(* Logix 5000 project; controller GolfBall vendor 1 type 14 code 149 rev 36.12; software revision 36.03 *)

TASK MainTask (continuous, watchdog 500 ms) : MainProgram

MODULES
   Local : vendor 1 type 14 code 149 (Compact 0, rev 36.12)
       : 1769-IQ16 (Compact 2, rev 1.1, Input RPI 20 ms)
       : 1769-IQ16 (Compact 3, rev 3.1, Input RPI 20 ms)
      Relay : 1769-OB16 (Compact 4, rev 3.1, Output RPI 20 ms)
      Discrete_IO : Embedded (Compact 1, rev 3.1, Output RPI 20 ms)
END_MODULES

TYPE FAULTRECORD :   // Stores the MajorFaultRecord attribute or MinorFaultRecord attribute of the Program object
STRUCT
   Time_Low : DINT;   // Lower 32 bits of the fault timestamp value
   Time_High : DINT;   // Upper 32 bits of the fault timestamp value
   Type : INT;   // Fault type (program, I/O, and so forth)
   Code : INT;   // Unique code for the fault
   Info : DINT[8];   // Fault specific information
END_STRUCT
END_TYPE

VAR_GLOBAL   (* controller tags *)
   Actuate_T1_Diverter : ALIAS FOR Local:4:O.Data.5; {access Read Only}
   Actuate_T1_Drop_Advance : ALIAS FOR Local:4:O.Data.12; {access Read Only}
   Actuate_T1_Drop_Release : ALIAS FOR Local:4:O.Data.13; {access Read Only}
   Actuate_T2_Diverter : ALIAS FOR Local:4:O.Data.6; {access Read Only}
   Actuate_T2_Drop_Advance : ALIAS FOR Local:4:O.Data.10; {access Read Only}
   Actuate_T2_Drop_Release : ALIAS FOR Local:4:O.Data.11; {access Read Only}
   Actuate_T3_Diverter : ALIAS FOR Local:4:O.Data.7; {access Read Only}
   Actuate_T3_Drop_Advance : ALIAS FOR Local:4:O.Data.8; {access Read Only}
   Actuate_T3_Drop_Release : ALIAS FOR Local:4:O.Data.9; {access Read Only}
   All_Tubes_Full : BOOL; {access Read Only}
   Auto_Run_Enable : BOOL; {access Read Only}
   Ball_Bypass_Photo : ALIAS FOR Local:1:I.Data.3; {access Read Only}
   Ball_Feeder_Extended : ALIAS FOR Local:3:I.Data.8; {access Read Only}
   Ball_Feeder_Intermediate : ALIAS FOR Local:3:I.Data.9; {access Read Only}
   Ball_Feeder_Retracted : ALIAS FOR Local:3:I.Data.10; {access Read Only}
   Ball_Feeder_Retracted_Timer : FBD_TIMER := (PRE := 400, Reset := 1); {access Read Only}
   Ball_Feeder_Step : DINT; {access Read Only}
   Ball_Present_Ball_Feeder : ALIAS FOR Local:3:I.Data.11; {access Read Only}
   Blink_Bit : BOOL; {access Read Only}
   Color : DINT; {access Read Only}
   Color_Advance_Cylinder_Extended : ALIAS FOR Local:1:I.Data.6; {access Read Only}
   Color_Advance_Cylinder_Retracted : ALIAS FOR Local:1:I.Data.7; {access Read Only}
   Color_Read_Advance_Cylinder_Timer : FBD_TIMER := (PRE := 1000); {access Read Only}
   Color_Read_Dwell_Timer : FBD_TIMER := (PRE := 1500); {access Read Only}
   Color_Release_Cylinder_Extended : ALIAS FOR Local:1:I.Data.8; {access Read Only}
   Color_Release_Cylinder_Retracted : ALIAS FOR Local:1:I.Data.9; {access Read Only}
   Color_Scan_Green : ALIAS FOR Local:3:I.Data.13; {access Read Only}
   Color_Scan_Orange : ALIAS FOR Local:3:I.Data.14; {access Read Only}
   Color_Scan_Pink : ALIAS FOR Local:3:I.Data.12; {access Read Only}
   Color_Sort_Dwell_Timer : FBD_TIMER := (TimerEnable := 1, PRE := 3500, ACC := 651, EN := 1, TT := 1); {access Read Only}
   Color_Sort_Step : DINT; {access Read Only}
   Drop_Ball_Feeder : ALIAS FOR Local:4:O.Data.15; {access Read Only}
   Dropping_Ball_Feeder : BOOL; {access Read Only}
   Fault : BOOL; {access Read Only}   // Master Fault
   Fault_Blink : BOOL; {access Read Only}
   Fault_Feeder_Drop_Timeout : BOOL; {access Read Only}
   Fault_Feeder_Lift_Timeout : BOOL; {access Read Only}
   Fault_Feeder_Watchdog : BOOL; {access Read Only}
   Feed_Bypass : BOOL; {access Read Only}
   Feed_Resume_OS : BOOL; {access Read Only}
   Feed_Resume_Storage : BOOL; {access Read Only}
   Feed_Run : BOOL; {access Read Only}
   Feeder_Drop_Timeout_Timer : FBD_TIMER := (PRE := 3000, Reset := 1); {access Read Only}
   Feeder_Extend_Count : DINT; {access Read Only}
   Feeder_Fault : BOOL; {access Read Only}
   Feeder_Fault_Active : BOOL; {access Read Only}
   Feeder_Hard_Fault_HMI : BOOL; {access Read Only}
   Feeder_Homing : BOOL; {access Read Only}
   Feeder_Lift_Timeout_Timer : FBD_TIMER := (TimerEnable := 1, PRE := 3000, ACC := 3000, EN := 1, DN := 1); {access Read Only}
   Feeder_Motion_Detected_OS : BOOL; {access Read Only}
   Feeder_Motion_Storage : BOOL; {access Read Only}
   Feeder_Recovery_Attempt_Counter : DINT; {access Read Only}
   Feeder_Recovery_Timer : FBD_TIMER := (PRE := 5000); {access Read Only}
   Feeder_Recovery_Total : DINT; {access Read Only}
   Feeder_Stuck_at_Sensor : BOOL; {access Read Only}
   Feeder_Watchdog_Timer : FBD_TIMER := (TimerEnable := 1, PRE := 5000, ACC := 3002, EN := 1, TT := 1); {access Read Only}
   Fill_Indexes_Cleared : BOOL := 1; {access Read Only}
   Green : DINT := 3; {access Read Only}
   HMI_All_Tubes_Are_Empty : INT := 10;
   HMI_ColorStationAdv : BOOL;
   HMI_ColorStationRel : BOOL := 1;
   HMI_Diverter1 : BOOL;
   HMI_Diverter2 : BOOL;
   HMI_Diverter3 : BOOL;
   HMI_DropFeedCylinder : BOOL;
   HMI_Fault_Reset_PB : BOOL;
   HMI_Page_State : INT := 2;
   HMI_RaiseFeedCylinder : BOOL;
   HMI_RequestedMode : INT;   // 30: Auto 20: Manual 10: Recovery 0: Undefined
   HMI_Setup_Done : BOOL := 1;
   HMI_Setup_in_Progress : BOOL;
   HMI_Setup_Request : BOOL;
   HMI_T1Drop1 : BOOL;
   HMI_T1Enable : BOOL := 1;
   HMI_T1SortMode : DINT;
   HMI_T2Drop1 : BOOL;
   HMI_T2Enable : BOOL;
   HMI_T2SortMode : DINT := 3;
   HMI_T3Drop1 : BOOL;
   HMI_T3Enable : BOOL;
   HMI_T3SortMode : DINT := 2;
   HMI_Trigger_Init : BOOL;
   HMI_Tube1_Diverter : BOOL;
   HMI_Tube2_Diverter : BOOL;
   HMI_Tube3_Diverter : BOOL;
   i : INT := 1; {access Read Only}
   idx1 : INT; {access Read Only}
   idx2 : INT; {access Read Only}
   idx3 : INT; {access Read Only}
   Lift_Ball_Feeder : ALIAS FOR Local:4:O.Data.14; {access Read Only}
   Lift_Time_Max : DINT; {access Read Only}
   Lift_Time_Max_Full : DINT; {access Read Only}
   Magazine_Full : ALIAS FOR Local:3:I.Data.15; {access Read Only}
   major_fault_record : FAULTRECORD := (Time_Low := -1123216650, Time_High := 209391, Info[0] := 16#ba69_35d2, Info[1] := 16#0003_31ef); {access Read Only}
   ModeChangeTimer : FBD_TIMER; {access Read Only}
   Number_of_Positions : DINT := 8;
   One_Sec_Blink_Timer : FBD_TIMER := (TimerEnable := 1, PRE := 500, ACC := 84, EN := 1, TT := 1); {access Read Only}
   Orange : DINT := 2; {access Read Only}
   Pink : DINT := 1; {access Read Only}
   PLC_Init_Done : BOOL := 1; {access Read Only}
   PowerUp_Handler_Ran : INT := 30; {access Read Only}
   Retract_Color_Advance_Cylinder : ALIAS FOR Local:4:O.Data.3; {access Read Only}
   Retract_Color_Release_Cylinder : ALIAS FOR Local:4:O.Data.4; {access Read Only}
   Run_Allowed : BOOL := 1; {access Read Only}
   Run_Latch : BOOL; {access Read Only}
   Run_Light : ALIAS FOR Local:4:O.Data.2; {access Read Only}
   Run_Permissive : BOOL; {access Read Only}
   Selected_Tube : DINT; {access Read Only}
   Sort_Bypass : BOOL; {access Read Only}
   Sort_Resume_OS : BOOL; {access Read Only}
   Sort_Resume_Storage : BOOL; {access Read Only}
   Sort_Run : BOOL; {access Read Only}
   Start_PB : ALIAS FOR Local:1:I.Data.5; {access Read Only}
   Start_PB_RE : BOOL; {access Read Only}
   Start_PB_Storage : BOOL; {access Read Only}
   Stop_PB : ALIAS FOR Local:1:I.Data.4; {access Read Only}
   System_Mode : DINT := 30; {access Read Only}   // 30: Auto 20: Manual 10: Recovery 0: Undefined
   System_Standby : BOOL := 1; {access Read Only}
   t : INT[3]; {access Read Only}
   T1_Color : INT[8] := ([0] := 3, [1] := 2, [2] := 1, [3] := 3, [4] := 2, [5] := 1, [6] := 3, [7] := 2); {access Read Only}
   T1_Diverter_Closed : ALIAS FOR Local:1:I.Data.11; {access Read Only}
   T1_Diverter_Opened : ALIAS FOR Local:1:I.Data.10; {access Read Only}
   T1_Drop_Adv_Cyl_Extended : ALIAS FOR Local:3:I.Data.4; {access Read Only}
   T1_Drop_Adv_Cyl_Retracted : ALIAS FOR Local:3:I.Data.5; {access Read Only}
   T1_Drop_Rel_Cyl_Extended : ALIAS FOR Local:3:I.Data.6; {access Read Only}
   T1_Drop_Rel_Cyl_Retracted : ALIAS FOR Local:3:I.Data.7; {access Read Only}
   T1_Index : DINT; {access Read Only}
   T1_TargetColor : INT := 3; {access Read Only}
   T1Full : BOOL; {access Read Only}
   T2_Color : INT[8] := ([0] := 3, [1] := 3, [2] := 3, [3] := 3, [4] := 3, [5] := 3, [6] := 3, [7] := 3); {access Read Only}
   T2_Diverter_Closed : ALIAS FOR Local:1:I.Data.13; {access Read Only}
   T2_Diverter_Opened : ALIAS FOR Local:1:I.Data.12; {access Read Only}
   T2_Drop_Adv_Cyl_Extended : ALIAS FOR Local:3:I.Data.0; {access Read Only}
   T2_Drop_Adv_Cyl_Retracted : ALIAS FOR Local:3:I.Data.1; {access Read Only}
   T2_Drop_Rel_Cyl_Extended : ALIAS FOR Local:3:I.Data.2; {access Read Only}
   T2_Drop_Rel_Cyl_Retracted : ALIAS FOR Local:3:I.Data.3; {access Read Only}
   T2_Index : DINT; {access Read Only}
   T2_TargetColor : INT := 3; {access Read Only}
   T2Full : BOOL; {access Read Only}
   T3_Color : INT[8] := ([0] := 2, [1] := 2, [2] := 2, [3] := 2, [4] := 2, [5] := 2, [6] := 2, [7] := 2); {access Read Only}
   T3_Diverter_Closed : ALIAS FOR Local:1:I.Data.15; {access Read Only}
   T3_Diverter_Opened : ALIAS FOR Local:1:I.Data.14; {access Read Only}
   T3_Drop_Adv_Cyl_Extended : ALIAS FOR Local:2:I.Data.0; {access Read Only}
   T3_Drop_Adv_Cyl_Retracted : ALIAS FOR Local:2:I.Data.1; {access Read Only}
   T3_Drop_Rel_Cyl_Extended : ALIAS FOR Local:2:I.Data.2; {access Read Only}
   T3_Drop_Rel_Cyl_Retracted : ALIAS FOR Local:2:I.Data.3; {access Read Only}
   T3_Index : DINT; {access Read Only}
   T3_TargetColor : INT := 2; {access Read Only}
   T3Full : BOOL; {access Read Only}
   Tube_1_BDPhoto : ALIAS FOR Local:1:I.Data.0; {access Read Only}   // Unused
   Tube_2_BDPhoto : ALIAS FOR Local:1:I.Data.1; {access Read Only}   // Unused
   Tube_3_BDPhoto : ALIAS FOR Local:1:I.Data.2; {access Read Only}   // Unused
   Tube_Color : INT[3,8] := ([0,0] := 3, [0,1] := 2, [0,2] := 1, [0,3] := 3, [0,4] := 2, [0,5] := 1, [0,6] := 3, [0,7] := 2, [1,0] := 3, [1,1] := 3, [1,2] := 3, [1,3] := 3, [1,4] := 3, [1,5] := 3, [1,6] := 3, [1,7] := 3, [2,0] := 2, [2,1] := 2, [2,2] := 2, [2,3] := 2, [2,4] := 2, [2,5] := 2, [2,6] := 2, [2,7] := 2); {access Read Only}
   Tube_Fill_Index : INT[3];
   White : DINT; {access Read Only}
END_VAR

PROGRAM Initialize   (* main routine Initialization *)

ROUTINE Initialization   (* structured text *)
// Initialize Outputs and Flags
   GSV(Program,THIS,MajorFaultRecord,major_fault_record.Time_Low);
   		major_fault_record.Type := 0;
   		major_fault_record.Code := 0;
   		SSV(Program,THIS,MajorFaultRecord,major_fault_record.Time_Low);
   
   // FORCE SAFE OUTPUTS
   // -------------------------------
       Lift_Ball_Feeder := 0;
       Drop_Ball_Feeder := 0;
   
       Actuate_T1_Diverter := 0;
       Actuate_T2_Diverter := 0;
       Actuate_T3_Diverter := 0;
   
   	Actuate_T1_Drop_Advance := 0;
   	Actuate_T1_Drop_Release := 0;
   	Actuate_T2_Drop_Advance := 0;
   	Actuate_T2_Drop_Release := 0;
   	Actuate_T3_Drop_Advance := 0;
   	Actuate_T3_Drop_Release := 0;
   
       Retract_Color_Advance_Cylinder := 0;
       Retract_Color_Release_Cylinder := 0;
   
       Run_Light := 0;
   
       //  RESET MACHINE STATE
       // -------------------------------
       Run_Latch := 0;
   	System_Mode := 30;
       Feeder_Fault_Active := 0;
   	Feeder_Recovery_Attempt_Counter := 0;
       Feeder_Homing := 0;
   
       Ball_Feeder_Step := 0;     // start in recovery/home
       Color_Sort_Step := 0;
   
       // CLEAR FAULTS
       // -------------------------------
       Fault_Feeder_Drop_Timeout := 0;
       Fault_Feeder_Lift_Timeout := 0;
       Fault_Feeder_Watchdog := 0;
   
       // RESET INTERNAL FLAGS
       // -------------------------------
       Feeder_Extend_Count := 0;
       Start_PB_Storage := Start_PB;
       Blink_Bit := 0;
   	HMI_Setup_Done := 0;
   	HMI_Trigger_Init := 0;
   	Number_of_Positions := 8;
   	HMI_All_Tubes_Are_Empty := 0;
   	Fill_Indexes_Cleared := 0;
   
   	// REQUEST OPERATOR INPUT
   	// -------------------------------
   	HMI_Setup_Request := 1;
   
       // DONE (RUN ONLY ONCE)
       // -------------------------------
   	PLC_Init_Done := 1;
END_ROUTINE
END_PROGRAM

PROGRAM MainProgram   (* main routine MainRoutine *)

ROUTINE Auto_Feed   (* structured text *)
// Feeding cylinder step-based machine.
   //----// Resume handling: //----//
   IF Feed_Resume_OS THEN
       Ball_Feeder_Step        := 00;   // every return to auto re-homes, same as a Stop
       Feeder_Motion_Storage := Ball_Feeder_Retracted OR Ball_Feeder_Intermediate
                                  OR Ball_Feeder_Extended;   // no phantom edge on resume
   END_IF;
   
   //----// Motion one-shot: //----//
   Feeder_Motion_Detected_OS := (Ball_Feeder_Retracted OR Ball_Feeder_Intermediate OR Ball_Feeder_Extended)
                                     AND NOT Feeder_Motion_Storage;
   Feeder_Motion_Storage := Ball_Feeder_Retracted OR Ball_Feeder_Intermediate OR Ball_Feeder_Extended;
   
   //----// Lift timeout: //----//
   IF Feeder_Extend_Count < 5 THEN
       Feeder_Lift_Timeout_Timer.PRE := 4000;
   ELSE
       Feeder_Lift_Timeout_Timer.PRE := 6000;
   END_IF;
   Feeder_Lift_Timeout_Timer.TimerEnable := Lift_Ball_Feeder;
   Feeder_Lift_Timeout_Timer.Reset       := NOT Lift_Ball_Feeder OR Feed_Resume_OS;
   TONR(Feeder_Lift_Timeout_Timer);
   
   // Lift margin monitor: longest normal stroke of each type, in ms
   IF Ball_Feeder_Step = 10 THEN
       IF Feeder_Extend_Count < 5 THEN
           IF Feeder_Lift_Timeout_Timer.ACC > Lift_Time_Max THEN Lift_Time_Max := Feeder_Lift_Timeout_Timer.ACC; END_IF;
       ELSE
           IF Feeder_Lift_Timeout_Timer.ACC > Lift_Time_Max_Full THEN Lift_Time_Max_Full := Feeder_Lift_Timeout_Timer.ACC; END_IF;
       END_IF;
   END_IF;
   
   IF Feeder_Lift_Timeout_Timer.DN AND NOT Feeder_Motion_Detected_OS THEN
       Fault_Feeder_Lift_Timeout := 1;
   END_IF;
   
   //----// Drop timeout: //----//
   IF Feeder_Extend_Count < 5 THEN
       Feeder_Drop_Timeout_Timer.PRE := 3000;
   ELSE
       Feeder_Drop_Timeout_Timer.PRE := 5000;
   END_IF;
   Feeder_Drop_Timeout_Timer.TimerEnable := Drop_Ball_Feeder;
   Feeder_Drop_Timeout_Timer.Reset       := NOT Drop_Ball_Feeder OR Feed_Resume_OS;
   TONR(Feeder_Drop_Timeout_Timer);
   IF Feeder_Drop_Timeout_Timer.DN AND NOT Ball_Feeder_Retracted THEN
       Fault_Feeder_Drop_Timeout := 1;
   END_IF;
   
   //----// Recovery timer: //----//
   Feeder_Recovery_Timer.TimerEnable := (Ball_Feeder_Step = 00);
   Feeder_Recovery_Timer.Reset       := Ball_Feeder_Retracted OR Feed_Resume_OS;
   Feeder_Recovery_Timer.PRE         := 5000;
   TONR(Feeder_Recovery_Timer);
   
   //----// Watchdog: //----//
   Feeder_Watchdog_Timer.TimerEnable := (Lift_Ball_Feeder OR Drop_Ball_Feeder) AND (Ball_Feeder_Step <> 00);
   Feeder_Watchdog_Timer.Reset       := Feeder_Motion_Detected_OS OR Feed_Resume_OS;
   Feeder_Watchdog_Timer.PRE         := 5000;
   TONR(Feeder_Watchdog_Timer);
   IF Feeder_Watchdog_Timer.DN THEN
       Fault_Feeder_Watchdog := 1;
   END_IF;
   
   //----// Feeder dropped dwell: //----//
   Ball_Feeder_Retracted_Timer.TimerEnable := Ball_Feeder_Retracted;
   Ball_Feeder_Retracted_Timer.Reset       := NOT Ball_Feeder_Retracted OR Feed_Resume_OS;
   Ball_Feeder_Retracted_Timer.PRE         := 400;
   TONR(Ball_Feeder_Retracted_Timer);
   
   //----------------// Recovery //---------------------//|
   	IF Feeder_Fault AND NOT Feeder_Fault_Active THEN
       	Feeder_Fault_Active := 1;
       	Ball_Feeder_Step := 00;
   	END_IF;
   
   
   
   CASE Ball_Feeder_Step OF
   	99:// HARD FAULT
   	// --------------------------------------------------
   
   		Lift_Ball_Feeder := 0;
   		Drop_Ball_Feeder := 0;
   		Feeder_Homing := 0;
   		Feeder_Hard_Fault_HMI := 1;    // Hard Fault flag to HMI
   
   		IF HMI_Fault_Reset_PB THEN
   			Ball_Feeder_Step := 00;    // Retry Recovery
   
   			Feeder_Fault_Active := 0;
   		END_IF;
   	00:// RECOVERY / INIT
   	// --------------------------------------------------
   
   		Lift_Ball_Feeder := 0;
   	 	Drop_Ball_Feeder := 1;
   	 	Feeder_Homing := 1;
   
   
   		IF Ball_Feeder_Retracted THEN
   			Ball_Feeder_Step := 05;
   			Feeder_Hard_Fault_HMI := 0;
   			Fault_Feeder_Drop_Timeout := 0;
   			Fault_Feeder_Lift_Timeout := 0;
   			Fault_Feeder_Watchdog := 0;
   			Drop_Ball_Feeder := 0;
   			IF Feeder_Fault_Active THEN
   	    	Feeder_Recovery_Attempt_Counter := Feeder_Recovery_Attempt_Counter + 1;
   			Feeder_Recovery_Total := Feeder_Recovery_Total + 1;
   			END_IF;
   		ELSIF Feeder_Recovery_Timer.DN THEN
   			Ball_Feeder_Step := 99;
   		END_IF;
   	05:// WAIT FOR START
   	// --------------------------------------------------
   
       	Lift_Ball_Feeder := 0;
       	Drop_Ball_Feeder := 0;
   		Feeder_Homing := 0;
   		Feeder_Fault_Active := 0;
       	IF Run_Latch AND NOT Magazine_Full THEN
           	Ball_Feeder_Step := 10;
       	END_IF;
   
   	10:// LIFT FEED CYLINDER
   	// --------------------------------------------------
   
       	Lift_Ball_Feeder := 1;
       	Drop_Ball_Feeder := 0;
       	IF Feeder_Extend_Count < 5 THEN
   
           	IF Ball_Feeder_Intermediate OR Ball_Feeder_Extended THEN
               	Ball_Feeder_Step := 20;
   				Feeder_Recovery_Attempt_Counter := 0;
           	END_IF;
   
       	ELSE
           	IF Ball_Feeder_Extended THEN
               	Ball_Feeder_Step := 20;
               	Feeder_Extend_Count := 0;
   				Feeder_Recovery_Attempt_Counter := 0;
           	END_IF;
       	END_IF;
   
   	20:// DROP FEED CYLINDER
   	// --------------------------------------------------
   
       	Lift_Ball_Feeder := 0;
       	Drop_Ball_Feeder := 1;
       	IF Ball_Feeder_Retracted THEN
           	Ball_Feeder_Step := 25;
       	END_IF;
   
   	25:// FEED CYLINDER DWELL
   	// --------------------------------------------------
   
   		IF Ball_Feeder_Retracted_Timer.DN THEN
   			Ball_Feeder_Step := 30;
   		END_IF;
   
   	30:// CYCLE COMPLETE / LOOP
   	// --------------------------------------------------
       	IF Magazine_Full THEN
           	Lift_Ball_Feeder := 0;
           	Drop_Ball_Feeder := 0;
           	Ball_Feeder_Step := 0;
           	Feeder_Extend_Count := 0;
   
       	ELSE
          	 	Feeder_Extend_Count := Feeder_Extend_Count + 1;
           	Ball_Feeder_Step := 05;
       	END_IF;
   
   END_CASE;
END_ROUTINE

ROUTINE Auto_Sort   (* structured text *)
// Sorting step-based machine.
   //----// Resume handling: //----//
   IF Sort_Resume_OS THEN
       Color_Sort_Step := 0;   // every return to auto restarts the sort cycle
   END_IF;
   
   //----// Timers: //----//
   Color_Read_Advance_Cylinder_Timer.TimerEnable := (Color_Sort_Step = 5);
   Color_Read_Advance_Cylinder_Timer.PRE         := 1000;
   TONR(Color_Read_Advance_Cylinder_Timer);
   
   Color_Read_Dwell_Timer.TimerEnable := (Color_Sort_Step = 10);
   Color_Read_Dwell_Timer.PRE         := 1500;
   TONR(Color_Read_Dwell_Timer);
   
   Color_Sort_Dwell_Timer.TimerEnable := (Color_Sort_Step = 30);
   CASE Selected_Tube OF
       1: Color_Sort_Dwell_Timer.PRE := 1500;
       2: Color_Sort_Dwell_Timer.PRE := 2200;
       3: Color_Sort_Dwell_Timer.PRE := 3200;
   ELSE
       Color_Sort_Dwell_Timer.PRE := 3500;
   END_CASE;
   TONR(Color_Sort_Dwell_Timer);
   
   CASE Color_Sort_Step OF
   	0: //INIT
   	// --------------------------------------------------
   		Actuate_T1_Diverter := 0;
   		Actuate_T2_Diverter := 0;
   		Actuate_T3_Diverter := 0;
   		Retract_Color_Release_Cylinder := 0;
   		Retract_Color_Advance_Cylinder := 0;
   
   		Color_Sort_Step := 5;
   
   	5: //ADVANCE
   	// --------------------------------------------------
   			Retract_Color_Release_Cylinder := 0;
   			Retract_Color_Advance_Cylinder := 1;
   		IF Color_Scan_Pink THEN
       		Color := Pink;
   		ELSIF Color_Scan_Orange THEN
       		Color := Orange;
   		ELSIF Color_Scan_Green THEN
       		Color := Green;
   		ELSE
       		Color := White;
   		END_IF;
   		IF Color_Read_Advance_Cylinder_Timer.DN THEN
   			Color_Sort_Step := 10;
   			Retract_Color_Advance_Cylinder := 0;
   		END_IF;
   
   	10: //TUBE SELECT
   	// --------------------------------------------------
   		IF Color_Read_Dwell_Timer.DN THEN
   			IF ((Color = T1_TargetColor) AND NOT T1Full) THEN
   				Selected_Tube := 1;
   
   			ELSIF ((Color = T2_TargetColor) AND NOT T2Full) THEN
   				Selected_Tube := 2;
   
   			ELSIF ((Color = T3_TargetColor) AND NOT T3Full) THEN
   				Selected_Tube := 3;
   
   			ELSE
   				Selected_Tube := 0;
   			END_IF;
   
   		Color_Sort_Step := 20;
   		END_IF;
   
   	20: //DIVERTER FIRE
   	// --------------------------------------------------
   		CASE Selected_Tube OF
   			0:
   				Actuate_T1_Diverter := 0;
   				Actuate_T2_Diverter := 0;
   				Actuate_T3_Diverter := 0;
   			1:
   				Actuate_T1_Diverter := 1;
   				Actuate_T2_Diverter := 0;
   				Actuate_T3_Diverter := 0;
   				Tube_Fill_Index[0] := Tube_Fill_Index[0] + 1;
   			2:
   				Actuate_T1_Diverter := 0;
   				Actuate_T2_Diverter := 1;
   				Actuate_T3_Diverter := 0;
   				Tube_Fill_Index[1] := Tube_Fill_Index[1] + 1;
   			3:
   				Actuate_T1_Diverter := 0;
   				Actuate_T2_Diverter := 0;
   				Actuate_T3_Diverter := 1;
   				Tube_Fill_Index[2] := Tube_Fill_Index[2] + 1;
   		END_CASE;
   
   		Color_Sort_Step := 30;
   
   	30: //RELEASE
   	// --------------------------------------------------
   		Retract_Color_Release_Cylinder := 1;
   
   		IF Color_Sort_Dwell_Timer.DN THEN Color_Sort_Step := 0;
   		END_IF;
   
   END_CASE;
END_ROUTINE

ROUTINE Color_Indexing   (* structured text *)
// Sorting Array Generation
   Pink := 1;
   Orange := 2;
   Green := 3;
   White := 0;
   
   // Sort modes: 0 = manual (the HMI writes each position of T<N>_Color),
   // 1-3 = fill all eight positions with Pink, Orange, or Green.
   IF (HMI_T1SortMode > 0) THEN
       FOR i := 0 TO 7 DO
           T1_Color[i] := HMI_T1SortMode;
       END_FOR;
   END_IF;
   IF (HMI_T2SortMode > 0) THEN
       FOR i := 0 TO 7 DO
           T2_Color[i] := HMI_T2SortMode;
       END_FOR;
   END_IF;
   IF (HMI_T3SortMode > 0) THEN
       FOR i := 0 TO 7 DO
           T3_Color[i] := HMI_T3SortMode;
       END_FOR;
   END_IF;
   
   // Each tube's target is the color assigned to its next empty position.
   // A full tube has no next position, so its target is -1, which no ball can match.
   // Logix won't accept an array element as a subscript; each fill count
   // writes into an INT first.
   idx1 := Tube_Fill_Index[0];
   idx2 := Tube_Fill_Index[1];
   idx3 := Tube_Fill_Index[2];
   
   IF (T1Full OR (idx1 < 0) OR (idx1 > 7)) THEN
       T1_TargetColor := -1;
   ELSE
       T1_TargetColor := T1_Color[idx1];
   END_IF;
   
   IF (T2Full OR (idx2 < 0) OR (idx2 > 7)) THEN
       T2_TargetColor := -1;
   ELSE
       T2_TargetColor := T2_Color[idx2];
   END_IF;
   
   IF (T3Full OR (idx3 < 0) OR (idx3 > 7)) THEN
       T3_TargetColor := -1;
   ELSE
       T3_TargetColor := T3_Color[idx3];
   END_IF;
END_ROUTINE

ROUTINE FaultRecovery   (* structured text *)
   
END_ROUTINE

ROUTINE Feed_ProcessBypass   (* structured text *)
// Homes feeding cylinder and disables feed process.
   Lift_Ball_Feeder := 0;
   IF NOT Ball_Feeder_Retracted THEN
   	Drop_Ball_Feeder := 1;
   ELSE
   	Drop_Ball_Feeder := 0;
   END_IF;
END_ROUTINE

ROUTINE Initialization   (* structured text *)
// Same as Power-Up Handler Initialization routine.
   // FORCE SAFE OUTPUTS
   // -------------------------------
       Lift_Ball_Feeder := 0;
       Drop_Ball_Feeder := 0;
   
       Actuate_T1_Diverter := 0;
       Actuate_T2_Diverter := 0;
       Actuate_T3_Diverter := 0;
   
   	Actuate_T1_Drop_Advance := 0;
   	Actuate_T1_Drop_Release := 0;
   	Actuate_T2_Drop_Advance := 0;
   	Actuate_T2_Drop_Release := 0;
   	Actuate_T3_Drop_Advance := 0;
   	Actuate_T3_Drop_Release := 0;
   
       Retract_Color_Advance_Cylinder := 0;
       Retract_Color_Release_Cylinder := 0;
   
       Run_Light := 0;
   
       //  RESET MACHINE STATE
       // -------------------------------
       Run_Latch := 0;
   	System_Mode := 30;
       Feeder_Fault_Active := 0;
   	Feeder_Recovery_Attempt_Counter := 0;
       Feeder_Homing := 0;
   
       Ball_Feeder_Step := 0;     // start in recovery/home
       Color_Sort_Step := 0;
   
       // CLEAR FAULTS
       // -------------------------------
       Fault_Feeder_Drop_Timeout := 0;
       Fault_Feeder_Lift_Timeout := 0;
       Fault_Feeder_Watchdog := 0;
   
       // RESET INTERNAL FLAGS
       // -------------------------------
       Feeder_Extend_Count := 0;
       Start_PB_Storage := Start_PB;
       Blink_Bit := 0;
   	HMI_Setup_Done := 0;
   	HMI_Trigger_Init := 0;
   	Number_of_Positions := 8;
   	HMI_All_Tubes_Are_Empty := 0;
   	Fill_Indexes_Cleared := 0;
   
   	// REQUEST OPERATOR INPUT
   	// -------------------------------
   	HMI_Setup_Request := 1;
   
       // DONE (RUN ONLY ONCE)
       // -------------------------------
   	PLC_Init_Done := 1;
END_ROUTINE

ROUTINE MainRoutine   (* ladder *)
// Executes subroutine calls.
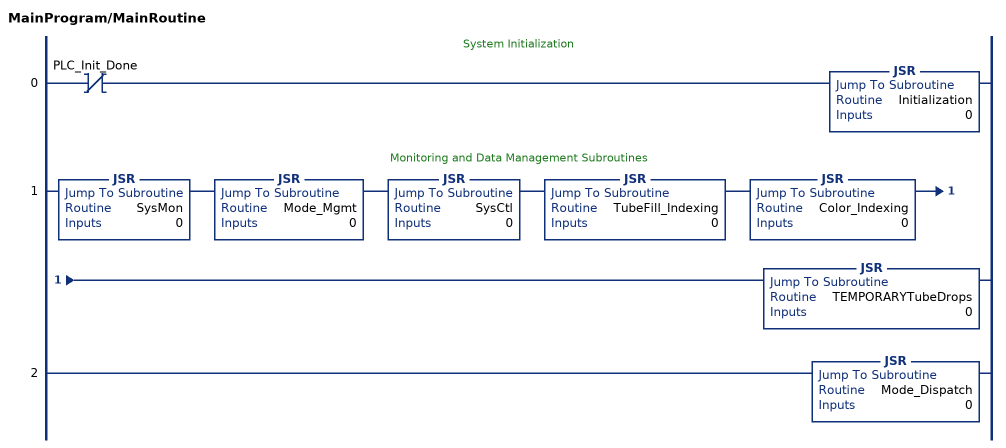
   // System Initialization
   0: XIO(PLC_Init_Done)JSR(Initialization,0);
   // Monitoring and Data Management Subroutines
   1: JSR(SysMon,0)JSR(Mode_Mgmt,0)JSR(SysCtl,0)JSR(TubeFill_Indexing,0)JSR(Color_Indexing,0)JSR(TEMPORARYTubeDrops,0);
   2: JSR(Mode_Dispatch,0);
END_ROUTINE

ROUTINE Manual_Ctrl   (* structured text *)
   	Lift_Ball_Feeder := HMI_RaiseFeedCylinder AND NOT Ball_Feeder_Extended;
   	Drop_Ball_Feeder := HMI_DropFeedCylinder AND NOT Ball_Feeder_Retracted;
   	Actuate_T1_Diverter := HMI_Diverter1;
   	Actuate_T2_Diverter := HMI_Diverter2;
   	Actuate_T3_Diverter := HMI_Diverter3;
   	Retract_Color_Advance_Cylinder := HMI_ColorStationAdv;
   	Retract_Color_Release_Cylinder := HMI_ColorStationRel;
END_ROUTINE

ROUTINE Mode_Dispatch   (* structured text *)
   // Stop request handler: (Auto only)
   IF ((NOT Run_Latch OR NOT Stop_PB) AND (System_Mode = 30)) THEN
       JSR(StopProcedures, 0);
   END_IF;
   
   Auto_Run_Enable := (Run_Latch AND PLC_Init_Done AND (System_Mode = 30));
   
   // Feed:
   Feed_Run            := (Auto_Run_Enable AND NOT Feed_Bypass);
   Feed_Resume_OS      := (Feed_Run AND NOT Feed_Resume_Storage);
   Feed_Resume_Storage := Feed_Run;
   IF Feed_Run THEN
       JSR(Auto_Feed, 0);
   ELSIF Auto_Run_Enable THEN        // Auto with Feed_Bypass on
       JSR(Feed_ProcessBypass, 0);
   END_IF;
   
   // Sort:
   Sort_Run            := (Auto_Run_Enable AND NOT Sort_Bypass);
   Sort_Resume_OS      := (Sort_Run AND NOT Sort_Resume_Storage);
   Sort_Resume_Storage := Sort_Run;
   IF Sort_Run THEN
       JSR(Auto_Sort, 0);
   ELSIF Auto_Run_Enable THEN        // Auto with Sort_Bypass on
       JSR(Sort_ProcessBypass, 0);
   END_IF;
   
   // Manual and recovery:
   IF (PLC_Init_Done AND (System_Mode = 20)) THEN
       JSR(Manual_Ctrl, 0);
   END_IF;
   IF (PLC_Init_Done AND (System_Mode = 10)) THEN
       JSR(FaultRecovery, 0);
   END_IF;
END_ROUTINE

ROUTINE Mode_Mgmt   (* structured text *)
// Mode Selection
   ModeChangeTimer.TimerEnable := ((HMI_RequestedMode <> System_Mode) AND (HMI_RequestedMode = 20));
   ModeChangeTimer.Reset := (HMI_RequestedMode = System_Mode);
   TONR(ModeChangeTimer);
   
   IF (HMI_RequestedMode <> System_Mode) THEN
   	//Auto
   	IF (HMI_RequestedMode = 30) THEN
   		System_Mode := HMI_RequestedMode;
   	END_IF;
   	//Manual
   	IF (HMI_RequestedMode = 20) THEN
   		JSR(StopProcedures, 0);
   		IF (ModeChangeTimer.DN AND NOT Dropping_Ball_Feeder) THEN
   			System_Mode := HMI_RequestedMode;
   		END_IF;
   	END_IF;
   END_IF;
END_ROUTINE

ROUTINE Sort_ProcessBypass   (* structured text *)
// Holds sort cylinders open and disables sort process.
   Actuate_T1_Diverter := 0;
   Actuate_T2_Diverter := 0;
   Actuate_T3_Diverter := 0;
   Retract_Color_Advance_Cylinder := 1;
   Retract_Color_Release_Cylinder := 1;
END_ROUTINE

ROUTINE StopProcedures   (* structured text *)
   Ball_Feeder_Step := 00;
   Lift_Ball_Feeder := 0;
   IF NOT Ball_Feeder_Retracted THEN
   	Dropping_Ball_Feeder := 1;
   	Drop_Ball_Feeder := 1;
   ELSE
   	Drop_Ball_Feeder := 0;
   END_IF;
   
   Color_Sort_Step := 0;
   Retract_Color_Advance_Cylinder := 0;
   Retract_Color_Release_Cylinder := 0;
   
   Actuate_T1_Diverter := 0;
   Actuate_T2_Diverter := 0;
   Actuate_T3_Diverter := 0;
END_ROUTINE

ROUTINE SysCtl   (* structured text *)
// System Control
   Start_PB_RE := (Start_PB AND NOT Start_PB_Storage);
   Start_PB_Storage := Start_PB;
   
   Run_Latch := ((Run_Latch OR Start_PB_RE) AND Stop_PB AND NOT Fault AND (System_Mode = 30));
   
   IF Fault THEN                                                                //Run Light
   	Run_Light := Fault_Blink;
   ELSE
   	Run_Light := Run_Latch;
   END_IF;
   
   
   Feeder_Stuck_at_Sensor := (Feeder_Recovery_Attempt_Counter > 3);
   Feeder_Fault :=                                                              //Feeder Fault Conditions
       Fault_Feeder_Drop_Timeout OR
   	Fault_Feeder_Lift_Timeout OR
   	Fault_Feeder_Watchdog;
   
   Fault := ((Feeder_Stuck_at_Sensor OR Feeder_Fault) AND NOT Feeder_Homing);
   
   IF HMI_Fault_Reset_PB THEN                                                       //Fault Reset
   	Fault_Feeder_Drop_Timeout := 0;
   	Fault_Feeder_Lift_Timeout := 0;
   	Fault_Feeder_Watchdog := 0;
   	Feeder_Stuck_at_Sensor := 0;
   	Feeder_Recovery_Attempt_Counter := 0;
   END_IF;
   
   // Bypass only after the current ball finishes (sort back at step 0),
   // Drop out as soon as any tube has room again.
   Sort_Bypass := (All_Tubes_Full AND (Sort_Bypass OR (Color_Sort_Step = 0)));
END_ROUTINE

ROUTINE SysMon   (* structured text *)
// System Monitoring
   //                                NOTES:
   //			HMI_Page_State (s) are: 1-Init; 2-Home; 3-Config; 4-Manual
   
   IF HMI_Trigger_Init THEN
   	PLC_Init_Done := 0;
   END_IF;
   IF (HMI_Page_State = 1) THEN
   	HMI_Setup_Request := 0;
   END_IF;
   
   Run_Allowed := Stop_PB AND HMI_Setup_Done AND PLC_Init_Done AND NOT Fault;
   System_Standby := Run_Allowed AND NOT Run_Latch;
   
   Fault_Blink := (Fault AND Blink_Bit);                                        //Fault Blink
   
   //----// Global 1Hz Blink Timer //----//|
   One_Sec_Blink_Timer.TimerEnable := 1;
   One_Sec_Blink_Timer.PRE := 500;
   TONR(One_Sec_Blink_Timer);
   IF One_Sec_Blink_Timer.DN THEN
   	One_Sec_Blink_Timer.Reset := 1;
   	Blink_Bit := NOT Blink_Bit;
   ELSE
   	One_Sec_Blink_Timer.Reset := 0;
   END_IF;
   //------------------------------------//|
   
   IF (T1Full AND T2Full AND T3Full) THEN
   	All_Tubes_Full := 1;
   ELSE
   	All_Tubes_Full := 0;
   END_IF;
   
   IF Drop_Ball_Feeder THEN
   	Dropping_Ball_Feeder := 1;
   ELSE
   	Dropping_Ball_Feeder := 0;
   END_IF;
END_ROUTINE

ROUTINE TEMPORARYTubeDrops   (* structured text *)
// To be replaced by tube emptying + ball shuffling subroutine(s)
   // Close Tube Drops (TEMPORARY)
   IF Run_Latch THEN
   	Actuate_T1_Drop_Advance := 0;
   	Actuate_T1_Drop_Release := 1;
   	Actuate_T2_Drop_Advance := 0;
   	Actuate_T2_Drop_Release := 1;
   	Actuate_T3_Drop_Advance := 0;
   	Actuate_T3_Drop_Release := 1;
   END_IF;
END_ROUTINE

ROUTINE TubeFill_Indexing   (* structured text *)
// Capacity Array Generation
   //                                NOTES:
   //			HMI_All_Tubes_Are_Empty States: 0-UNDEF; 10-Yes; 20-No;
   
   IF ((HMI_All_Tubes_Are_Empty = 10) AND NOT Fill_Indexes_Cleared) THEN
   Tube_Fill_Index[0] := 0;
   Tube_Fill_Index[1] := 0;
   Tube_Fill_Index[2] := 0;
   Fill_Indexes_Cleared := 1;
   END_IF;
   
   T1Full := (Tube_Fill_Index[0] >= Number_of_Positions);
   T2Full := (Tube_Fill_Index[1] >= Number_of_Positions);
   T3Full := (Tube_Fill_Index[2] >= Number_of_Positions);
   //Clamp
   IF (Tube_Fill_Index[0] > Number_of_Positions) THEN
   	Tube_Fill_Index[0] := Number_of_Positions;
   END_IF;
   IF (Tube_Fill_Index[1] > Number_of_Positions) THEN
   	Tube_Fill_Index[1] := Number_of_Positions;
   END_IF;
   IF (Tube_Fill_Index[2] > Number_of_Positions) THEN
   	Tube_Fill_Index[2] := Number_of_Positions;
   END_IF;
END_ROUTINE
END_PROGRAM
